FUNCTION_BLOCK TestFB
VAR_INPUT
	//Test inputs
	command_StartTest : BOOL;
	command_StopTest  : BOOL;
	command_Reset     : BOOL;
	command_StartSeed : BOOL;
END_VAR
VAR_OUTPUT
	errorDiagMsg		: STRING(255);
END_VAR
VAR
	bStartup          : BOOL  := TRUE;
	methaneStartUpDelay		: TON;
	methaneSettingTime		: TON;
	ignitionTimer       	: TON;
	ignitionDelay 			: TON;
	ignitionCheckTimer		: TON;
	testTimer				: TON;
END_VAR

CASE gMachine.testCell.state OF
	TEST_STATE.STARTUP:
		IF bStartup THEN
			bStartup := FALSE;
			gMachine.testCell.TSIG_ZVSIgnite(Init:=FALSE, pIO:=ADR(gIO.DO_ZVSIgnite));
			gMachine.testCell.TSIG_CombustorAirSolenoid(Init:=FALSE, pIO:=ADR(gIO.DO_CombustorAirSolenoid));   
			gMachine.testCell.TSIG_MethaneSolenoid(Init:=FALSE, pIO:=ADR(gIO.DO_MethaneSolenoid));      
			gMachine.testCell.TSIG_WaterQuenchSolenoid(Init:=FALSE, pIO:=ADR(gIO.DO_WaterQuenchSolenoid));  
			gMachine.testCell.TSIG_SeederExtendSolenoid(Init:=FALSE, pIO:=ADR(gIO.DO_SeederExtendSolenoid));    
			gMachine.testCell.TSIG_SeederRetractSolenoid(Init:=FALSE, pIO:=ADR(gIO.DO_SeederRetractSolenoid));  
			gMachine.testCell.TSIG_FluidizationSolenoid(Init:=FALSE, pIO:=ADR(gIO.DO_SeederFluidization));   
			gMachine.testCell.TSIG_EjectorSolenoid(Init:=FALSE, pIO:=ADR(gIO.DO_EjectorSolenoid));     
			gMachine.testCell.state := TEST_STATE.IDLE;	
		END_IF
		
	TEST_STATE.IDLE:
		//Make sure all timers are reset from the idle state
		IF command_StartTest THEN
			command_StartTest := FALSE;
			gMachine.testCell.state := TEST_STATE.CHECK_TEST_READY;
		END_IF
		
	TEST_STATE.CHECK_TEST_READY:
		gMachine.testCell.state := TEST_STATE.SET_TEST_VARIABLES;
		
	TEST_STATE.SET_TEST_VARIABLES:
		gMachine.testCell.state := TEST_STATE.START_TEST;
	TEST_STATE.START_TEST:
		gIO.DO_CollectData := TRUE;
		gIO.DO_CombustorAirSolenoid := TRUE;
		methaneStartUpDelay(IN:=TRUE, PT:=T#10S);
		IF methaneStartUpDelay.Q THEN
			IF gScaledIO.monitoredValues[1].scaledValue > gMachineSettings.safetyParameters.minAirPressure THEN
				methaneStartUpDelay(IN:=FALSE);
				gIO.DO_MethaneSolenoid := TRUE;
				gMachine.testCell.state := TEST_STATE.START_IGNITION;
			ELSE
				methaneStartUpDelay(IN:=FALSE);
				errorDiagMsg := 'Methane flow attempted without air';
				gMachine.testCell.state := TEST_STATE.ERROR;
			END_IF
		END_IF
	
	TEST_STATE.START_IGNITION:
		ignitionDelay(IN:=TRUE, PT:=T#1S);
		IF ignitionDelay.Q THEN
			IF gScaledIO.monitoredValues[2].scaledValue > gMachineSettings.safetyParameters.minMethanePressure THEN 
				gIO.DO_ZVSIgnite := TRUE;
				ignitionTimer(IN:=TRUE, PT:=T#1S);
				IF ignitionTimer.Q THEN
					gIO.DO_ZVSIgnite := FALSE;
					ignitionDelay(IN:=FALSE);
					ignitionTimer(IN:=FALSE);
					gMachine.testCell.state := TEST_STATE.CHECK_IGNITION;
				END_IF
			ELSE
				ignitionDelay(IN:=FALSE);
				ignitionTimer(IN:=FALSE);
				errorDiagMsg := 'Ignition Attempted Without Methane';
				gMachine.testCell.state := TEST_STATE.ERROR;	
			END_IF
		END_IF
		
	TEST_STATE.CHECK_IGNITION: 
		ignitionCheckTimer(IN:=TRUE, PT:=T#1S);
		IF ignitionCheckTimer.Q THEN
			ignitionCheckTimer(IN:=FALSE);
			IF gScaledIO.monitoredValues[7].scaledValue > gMachineSettings.safetyParameters.minCombustorPressure THEN
				gMachine.testCell.state := TEST_STATE.WAIT_FOR_SEED;	
			ELSE
				errorDiagMsg := 'Ignition failure, no combustion occured';
				gMachine.testCell.state := TEST_STATE.ERROR;	
			END_IF
		END_IF
	
	TEST_STATE.WAIT_FOR_SEED:
		IF command_StartSeed THEN
			gMachine.testCell.state := TEST_STATE.RUN_TEST;
		END_IF
		
	
	TEST_STATE.RUN_TEST:
		//Start time based systems
		testTimer(IN:=TRUE, PT:=MAX(gMachineSettings.testParameters.ZVSIgniteOffTime, 
									gMachineSettings.testParameters.MethaneSolenoidOffTime, 
									gMachineSettings.testParameters.SeederExtendSolenoidOffTime, 
									gMachineSettings.testParameters.FluidizationSolenoidOffTime));
		gMachine.testCell.TSIG_ZVSIgnite(Init:=TRUE, Start_Time:=gMachineSettings.testParameters.ZVSIgniteOnTime,End_Time:=gMachineSettings.testParameters.ZVSIgniteOffTime);
		gMachine.testCell.TSIG_MethaneSolenoid(Init:=TRUE, Start_Time:=gMachineSettings.testParameters.MethaneSolenoidOnTime, End_Time:=gMachineSettings.testParameters.MethaneSolenoidOffTime);
		gMachine.testCell.TSIG_SeederExtendSolenoid(Init:=TRUE, Start_Time:=gMachineSettings.testParameters.SeederExtendSolenoidOnTime, End_Time:=gMachineSettings.testParameters.SeederExtendSolenoidOffTime);
		gMachine.testCell.TSIG_FluidizationSolenoid(Init:=TRUE, Start_Time:=gMachineSettings.testParameters.FluidizationSolenoidOnTime, End_Time:=gMachineSettings.testParameters.FluidizationSolenoidOffTime);
	
		//run watchdog tests
		//IF gIO.DI_SeederExtendLimitSensor THEN
		//	testTimer(IN:=FALSE);
		//	gMachine.testCell.state := TEST_STATE.COMPLETE;
		//END_IF
		IF 	testTimer.Q THEN
			testTimer(IN:=FALSE);
			gMachine.testCell.state := TEST_STATE.COMPLETE;
		END_IF
		IF  gScaledIO.monitoredValues[1].scaledValue < gMachineSettings.safetyParameters.minAirPressure THEN
			errorDiagMsg := 'Loss of air pressure during testing'; 
			gMachine.testCell.state := TEST_STATE.ERROR;
		END_IF
		
		IF 	gScaledIO.monitoredValues[2].scaledValue < gMachineSettings.safetyParameters.minMethanePressure THEN
			errorDiagMsg := 'Loss of methane pressure during testing'; 
			gMachine.testCell.state := TEST_STATE.ERROR;
		END_IF
		
		IF 	gScaledIO.monitoredValues[7].scaledValue < gMachineSettings.safetyParameters.minCombustorPressure THEN
			errorDiagMsg := 'Loss of chamber pressure, unstarted engine';
			gMachine.testCell.state := TEST_STATE.ERROR;
		END_IF
		
		IF gScaledIO.monitoredValues[4].scaledValue < gMachineSettings.safetyParameters.minFacilityPressure THEN
			errorDiagMsg := 'Tank pressure too low during testing';
			gMachine.testCell.state := TEST_STATE.ERROR;
		END_IF
		
	TEST_STATE.COMPLETE:
		gMachine.testCell.TSIG_ZVSIgnite(Init:=FALSE);
		gMachine.testCell.TSIG_CombustorAirSolenoid(Init:=FALSE);   
		gMachine.testCell.TSIG_MethaneSolenoid(Init:=FALSE);      
		gMachine.testCell.TSIG_WaterQuenchSolenoid(Init:=FALSE);  
		gMachine.testCell.TSIG_SeederExtendSolenoid(Init:=FALSE);    
		gMachine.testCell.TSIG_SeederRetractSolenoid(Init:=FALSE);  
		gMachine.testCell.TSIG_FluidizationSolenoid(Init:=FALSE);   
		gMachine.testCell.TSIG_EjectorSolenoid(Init:=FALSE);     
	
	TEST_STATE.STOP:
		//reset timers
		gMachine.testCell.TSIG_ZVSIgnite(Init:=FALSE);
		gMachine.testCell.TSIG_CombustorAirSolenoid(Init:=FALSE);   
		gMachine.testCell.TSIG_MethaneSolenoid(Init:=FALSE);      
		gMachine.testCell.TSIG_WaterQuenchSolenoid(Init:=FALSE);  
		gMachine.testCell.TSIG_SeederExtendSolenoid(Init:=FALSE);    
		gMachine.testCell.TSIG_SeederRetractSolenoid(Init:=FALSE);  
		gMachine.testCell.TSIG_FluidizationSolenoid(Init:=FALSE);   
		gMachine.testCell.TSIG_EjectorSolenoid(Init:=FALSE);     
		gMachine.testCell.state := TEST_STATE.BLOWDOWN;
		//run purge air 
	TEST_STATE.BLOWDOWN:
		gMachine.testCell.TSIG_CombustorAirSolenoid(Init:=TRUE, Start_Time := INT_TO_TIME(0), End_Time := INT_TO_TIME(5000));
		gHMI.iBlowdownTimeProgress := REAL_TO_INT(TIME_TO_INT(gMachine.testCell.TSIG_CombustorAirSolenoid.ET - gMachine.testCell.TSIG_CombustorAirSolenoid.Start_Time) * (100) / TIME_TO_INT(gMachine.testCell.TSIG_CombustorAirSolenoid.End_Time - gMachine.testCell.TSIG_CombustorAirSolenoid.Start_Time));
		IF NOT gMachine.testCell.TSIG_CombustorAirSolenoid.Q THEN
			gMachine.testCell.state := TEST_STATE.BLOWDOWN_COMPLETE;
		END_IF
	TEST_STATE.BLOWDOWN_COMPLETE:
		gMachine.testCell.TSIG_CombustorAirSolenoid(Init:=FALSE);
		gHMI.iBlowdownTimeProgress := 0;
		gMachine.testCell.state := TEST_STATE.IDLE;
		
	TEST_STATE.ESTOP: 
		gMachine.testCell.TSIG_ZVSIgnite(Init:=FALSE);
		gMachine.testCell.TSIG_CombustorAirSolenoid(Init:=FALSE);   
		gMachine.testCell.TSIG_MethaneSolenoid(Init:=FALSE);      
		gMachine.testCell.TSIG_WaterQuenchSolenoid(Init:=FALSE);  
		gMachine.testCell.TSIG_SeederExtendSolenoid(Init:=FALSE);    
		gMachine.testCell.TSIG_SeederRetractSolenoid(Init:=FALSE);  
		gMachine.testCell.TSIG_FluidizationSolenoid(Init:=FALSE);   
		gMachine.testCell.TSIG_EjectorSolenoid(Init:=FALSE);    
		
		//reset IO
		gIO.DO_CombustorAirSolenoid := FALSE;
		gIO.DO_MethaneSolenoid := FALSE;
		gIO.DO_SeederExtendSolenoid := FALSE;
		gIO.DO_SeederFluidization := FALSE;
		gIO.DO_WaterQuenchSolenoid := FALSE;
		gIO.DO_ZVSIgnite := FALSE;
		gIO.DO_EjectorSolenoid := FALSE;
	
			
	TEST_STATE.WAIT_FOR_RESET:
		IF command_Reset THEN
			command_Reset := FALSE;
			gIO.DO_Reset  := TRUE;
			gMachine.testCell.state := TEST_STATE.RESETTING;
		END_IF
		
	TEST_STATE.RESETTING: 
		IF gIO.DI_24VAtSolenoids THEN
			gIO.DO_Reset := FALSE;
			gMachine.testCell.state := TEST_STATE.IDLE;
		END_IF	
	
	TEST_STATE.ERROR: 
		gMachine.testCell.state := TEST_STATE.STOP;
		
END_CASE

END_FUNCTION_BLOCK

(* stored: Version 1.1.0.1, ProductVersion 3.1.4024.12
   POU TestFB: Id {4ccabcbe-2adc-4f87-a510-41641d4b21c7}, SpecialFunc None *)
